{attribute 'qualified_only'}
VAR_GLOBAL
END_VAR

(* stored: Version 1.1.0.1, ProductVersion 3.1.4024.16
   GVL Testing_DB: Id {3d651cd0-c587-4c8c-b130-9112feba3e6a} *)
